INTERFACE I_Callback EXTENDS I_Subscriber

END_INTERFACE

(* stored: Version 1.1.0.1, ProductVersion 3.1.4024.11
   Itf I_Callback: Id {0d16a7d4-f9f7-4cbf-9242-6b59d0319774} *)
